KUKA KRL program: geek_test2.src

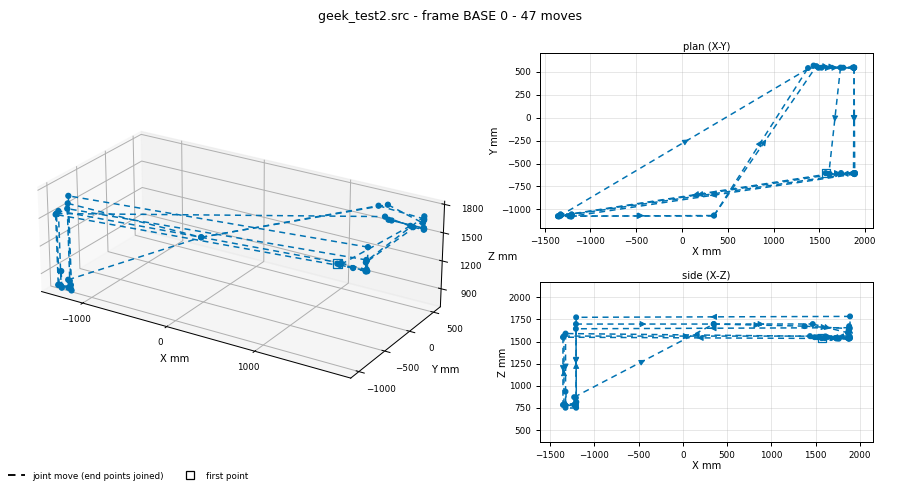
[picture p0: tool path of geek_test2.src in frame BASE 0, 47 of 50 moves have a stored position in this frame; points joined in program order, loops and branches not executed]
&ACCESS RVP
&REL 423
&PARAM TEMPLATE = C:\KRC\Roboter\Template\vorgabe
&PARAM EDITMASK = *
DEF geek_test2( )
INT I
;FOLD INI;%{PE}%V3.2.0,%MKUKATPBASIS,%CINIT,%VCOMMON,%P
;FOLD BAS INI;%{E}%V3.2.0,%MKUKATPBASIS,%CINIT,%VINIT,%P
GLOBAL INTERRUPT DECL 3 WHEN $STOPMESS==TRUE DO IR_STOPM ( )
INTERRUPT ON 3
BAS (#INITMOV,0 )
;ENDFOLD (BAS INI)
;FOLD A20 INI;%{E}%V3.2.0,%MKUKATPA20,%CINIT,%VINIT,%P
IF ARC20==TRUE THEN
A20 (ARC_INI)
INTERRUPT DECL 6 WHEN $CYCFLAG[3]==FALSE DO A20(TECH_STOP2)
ENDIF
;ENDFOLD (A20 INI)
;FOLD A10 INI;%{E}%V3.2.0,%MKUKATPARC,%CINIT,%VINIT,%P
IF A10_OPTION==#ACTIVE THEN
INTERRUPT DECL 4 WHEN $CYCFLAG[2]==FALSE DO A10 (#APPL_ERROR)
INTERRUPT DECL 7 WHEN A_ARC_SWI==#ACTIVE DO A10 (#ARC_SEAM)
INTERRUPT DECL 5 WHEN A_FLY_ARC==TRUE DO A10 (#HPU_ARC)
INTERRUPT  ON 5
A10_INI ( )
ENDIF
;ENDFOLD (A10 INI)
;FOLD GRIPPER INI;%{E}%V3.2.0,%MKUKATPGRIPPER,%CINIT,%VINIT,%P
USER_GRP(0,DUMMY,DUMMY,GDEFAULT)
;ENDFOLD (GRIPPER INI)
;FOLD SPOT INI;%{E}%V3.2.0,%MKUKATPSPOT,%CINIT,%VINIT,%P
USERSPOT(#INIT)
;ENDFOLD (SPOT INI)
;FOLD TOUCHSENSE INI;%{E}%V3.2.0,%MKUKATPTS,%CINIT,%VINIT,%P
IF H70_OPTION THEN
INTERRUPT DECL 15 WHEN $MEAS_PULSE[TOUCH_I[TOUCH_ACTIVE].IN_NR] DO H70 (6,CD0 )
INTERRUPT DECL 16 WHEN $ZERO_MOVE DO H70 (7,CD0 )
INTERRUPT DECL 17 WHEN $TECHPAR_C[FG_TOUCH,8]>0.5 DO H70 (8,CD0)
H70 (1,CD0 )
ENDIF
;ENDFOLD (TOUCHSENSE INI)
;FOLD USER INI;%{E}%V3.2.0,%MKUKATPUSER,%CINIT,%VINIT,%P
;Make your modifications here
;ENDFOLD (USER INI)
;ENDFOLD (INI)

;FOLD                                    (LOCAL DECLARATIONS)
FOR I=1 TO 6
$VEL_AXIS[I]=10
$ACC_AXIS[I]=2
ENDFOR

$TOOL=$NULLFRAME
$BASE=$NULLFRAME
$FILTER=$DEF_FLT_PTP
$LOAD.M=325
$LOAD.CM.X=100
$LOAD.CM.Y=0
$LOAD.CM.Z=300
$LOAD.CM.A=0
$LOAD.CM.B=0
$LOAD.CM.C=0
$APO.CPTP=80
$ADVANCE=5
;ENDFOLD

$VEL_AXIS[1]=100
$VEL_AXIS[2]=100
$VEL_AXIS[3]=100
$VEL_AXIS[4]=100
$VEL_AXIS[5]=100
$VEL_AXIS[6]=100

$ACC_AXIS[1]=100
$ACC_AXIS[2]=100
$ACC_AXIS[3]=100
$ACC_AXIS[4]=100
$ACC_AXIS[5]=100
$ACC_AXIS[6]=100

LOOP
PTP XHOME1
PTP {POS: X 1568.75, Y -604.56, Z 1539.05, A 176.81, B 5.23, C 179.57, S 2., T 10.}
PTP {POS: X 1889.33, Y -604.65, Z 1539.11, A 176.8, B 5.24, C 179.57, S 2., T 10.}
PTP {POS: X 1889.33, Y -604.66, Z 1784.88, A 176.8, B 5.24, C 179.57, S 2., T 10.}

PTP {POS: X -1205.3, Y -1056.67, Z 1774.53, A 176.8, B 5.24, C 179.57, S 2., T 10.}
PTP {POS: X -1205.31, Y -1056.67, Z 752.83, A 176.8, B 5.24, C 179.57, S 2., T 10.}
PTP {POS: X -1325.54, Y -1056.67, Z 752.83, A 176.8, B 5.24, C 179.57, S 2., T 10.}
PTP {POS: X -1325.54, Y -1056.67, Z 935.54, A 176.8, B 5.24, C 179.57, S 2., T 10.}
PTP XHOME1
PTP {POS: X 1523.57, Y 546.13, Z 1549.44, A 176.85, B 3.13, C 176.25, S 2., T 43.}
PTP {POS: X 1879.05, Y 546.12, Z 1549.45, A 176.85, B 3.13, C 176.25, S 2., T 43.}

PTP {POS: X 1879.05, Y 546.12, Z 1674.48, A 176.85, B 3.13, C 176.25, S 2., T 43.}
PTP {POS: X 1886.43, Y -611.96, Z 1649.53, A 176.85, B 3.13, C 176.25, S 2., T 10.}
PTP {POS: X 1886.42, Y -611.96, Z 1558.62, A 176.85, B 3.13, C 176.25, S 2., T 10.}
PTP {POS: X 1612.1, Y -611.95, Z 1558.62, A 176.85, B 3.13, C 176.25, S 2., T 10.}
PTP {POS: X -1324.79, Y -1068.2, Z 1591.08, A 177.19, B -1.41, C -177.29, S 2., T 10.}
PTP {POS: X -1324.81, Y -1068.21, Z 779.47, A 177.19, B -1.41, C -177.29, S 2., T 10.}
PTP {POS: X -1207.38, Y -1068.2, Z 779.46, A 177.19, B -1.41, C -177.29, S 2., T 10.}
PTP {POS: X -1203.08, Y -1068.17, Z 817.61, A 177.19, B -1.41, C -177.29, S 2., T 10.}

PTP {POS: X -1207.38, Y -1068.21, Z 1698.38, A 177.19, B -1.41, C -177.29, S 2., T 10.}
PTP {POS: X 349.36, Y -1068.21, Z 1698.37, A 177.19, B -1.41, C -177.29, S 2., T 2.}
PTP {POS: X 1468.03, Y 563.31, Z 1698.37, A 176.98, B 2.48, C 176.95, S 2., T 43.}
PTP {POS: X 1865.33, Y 547.83, Z 1599.94, A 176.97, B 2.48, C 176.95, S 2., T 43.}
PTP {POS: X 1882.14, Y 547.92, Z 1539.21, A 176.97, B 2.48, C 176.95, S 2., T 43.}
PTP {POS: X 1730.87, Y 547.9, Z 1539.21, A 176.97, B 2.48, C 176.95, S 2., T 43.}
PTP {POS: X 1603.1, Y -616.68, Z 1539.22, A 177.25, B 7.45, C 179.06, S 2., T 10.}
PTP {POS: X 1882.37, Y -616.08, Z 1541.92, A 177.25, B 7.46, C 179.06, S 2., T 10.}
PTP {POS: X 1882.37, Y -616.09, Z 1657.36, A 177.25, B 7.46, C 179.06, S 2., T 10.}
PTP {POS: X -1208.37, Y -1077.13, Z 1645.05, A 177.27, B 7.47, C 179.07, S 2., T 10.}
PTP {POS: X -1208.37, Y -1077.12, Z 865.12, A 177.75, B -1.58, C -177.07, S 2., T 10.}
PTP {POS: X -1208.39, Y -1077.13, Z 797.13, A 177.75, B -1.58, C -177.07, S 2., T 10.}
PTP {POS: X -1342.84, Y -1077.15, Z 790.23, A 177.74, B -1.58, C -177.07, S 2., T 10.}
PTP {POS: X -1342.83, Y -1077.15, Z 1562.32, A 177.74, B -1.58, C -177.07, S 2., T 10.}
PTP {POS: X 1436.76, Y 570.02, Z 1562.36, A 177.21, B 4.08, C 175.59, S 2., T 43.}
PTP {POS: X 1762.06, Y 546.43, Z 1532.7, A 177.19, B 4.09, C 175.59, S 2., T 43.}

PTP {POS: X 1878.41, Y 546.44, Z 1532.69, A 177.19, B 4.09, C 175.59, S 2., T 43.}

PTP {POS: X 1878.41, Y 546.45, Z 1633.71, A 177.19, B 4.09, C 175.59, S 2., T 43.}
PTP {POS: X 1873.05, Y -607.43, Z 1626.15, A 177.19, B 4.09, C 175.59, S 2., T 10.}
PTP {POS: X 1873.04, Y -607.43, Z 1534.85, A 177.19, B 4.09, C 175.59, S 2., T 10.}
PTP {POS: X 1736.94, Y -603.59, Z 1534.84, A 177.19, B 4.09, C 175.59, S 2., T 10.}
PTP {POS: X -1354.22, Y -1076.06, Z 1549.73, A 177.39, B -0.06, C -176.19, S 2., T 10.}
PTP {POS: X -1354.23, Y -1076.06, Z 784.67, A 177.39, B -0.06, C -176.19, S 2., T 10.}
PTP {POS: X -1227.53, Y -1076.05, Z 784.66, A 177.39, B -0.06, C -176.19, S 2., T 10.}

PTP {POS: X -1227.53, Y -1076.09, Z 872.3, A 177.39, B -0.07, C -176.19, S 2., T 10.}
PTP {POS: X 349.36, Y -1068.21, Z 1698.37, A 177.19, B -1.41, C -177.29, S 2., T 2.}
PTP {POS: X 1376.39, Y 542.37, Z 1674.57, A 177.39, B -0.07, C -176.19, S 2., T 35.}
PTP {POS: X 1878.45, Y 545.31, Z 1647.22, A 177.39, B -0.07, C -176.19, S 2., T 35.}
PTP {POS: X 1878.45, Y 545.3, Z 1549.83, A 177.27, B 0.99, C 177.31, S 2., T 43.}
PTP {POS: X 1489.95, Y 545.3, Z 1549.84, A 177.27, B 0.99, C 177.31, S 2., T 43.}



















PTP XHOME1

ENDLOOP
END
